{attribute 'call_after_init'}
{attribute 'reflection'}
FUNCTION_BLOCK ABSTRACT T_UnitTestBase IMPLEMENTS I_UnitTest
VAR
    {attribute 'instance-path'}
    {attribute 'no_init'}
    {attribute 'analysis' := '-33'} // Inhibit unused variable warning
    InstanceName : T_MaxString;     // Initialised with the instance name

    Project  : T_MaxString;
    Plc      : T_MaxString;
    TestName : T_MaxString;

    _TestCompleted : BOOL;
    _TestFailed    : BOOL;
    State          : INT;
    CycleCount     : UDINT;
    Retest         : BOOL;
END_VAR

METHOD AssertEquals_ANY : BOOL
VAR_INPUT
    Expected : ANY;
    Actual   : ANY;
    Message  : T_MaxString;
END_VAR
VAR
    ComparisonResult : DINT;
END_VAR
ComparisonResult := MEMCMP(pBuf1 := Expected.pValue,
                           pBuf2 := Actual.pValue,
                           n     := DINT_TO_UDINT(Actual.diSize));

IF Expected.TypeClass <> Actual.TypeClass THEN
    F_LogError(TestName, FormatStringEx1('Assertion Failed - %s', Message));
    TestFailed := TRUE;
    RETURN;

ELSIF Expected.diSize <> Actual.diSize THEN
    F_LogError(TestName, FormatStringEx1('Assertion Failed - %s', Message));
    TestFailed := TRUE;
    RETURN;

ELSIF ComparisonResult <> 0 THEN
    F_LogError(TestName, FormatStringEx1('Assertion Failed - %s', Message));
    TestFailed := TRUE;
    RETURN;
END_IF

AssertEquals_ANY := TRUE;
END_METHOD

METHOD AssertEquals_BOOL : BOOL
VAR_INPUT
    Expected : BOOL;
    Actual   : BOOL;
    Message  : T_MaxString;
END_VAR
IF Expected <> Actual THEN
    F_LogError(TestName, FormatStringEx1('Assertion Failed - %s', Message));
    TestFailed := TRUE;
    RETURN;
END_IF

AssertEquals_BOOL := TRUE;
END_METHOD

METHOD AssertEquals_BYTE : BOOL
VAR_INPUT
    Expected : BYTE;
    Actual   : BYTE;
    Message  : T_MaxString;
END_VAR
IF Expected <> Actual THEN
    F_LogError(TestName, FormatStringEx1('Assertion Failed - %s', Message));
    TestFailed := TRUE;
    RETURN;
END_IF

AssertEquals_BYTE := TRUE;
END_METHOD

METHOD AssertEquals_DINT : BOOL
VAR_INPUT
    Expected : DINT;
    Actual   : DINT;
    Message  : T_MaxString;
END_VAR
IF Expected <> Actual THEN
    F_LogError(TestName, FormatStringEx1('Assertion Failed - %s', Message));
    TestFailed := TRUE;
    RETURN;
END_IF

AssertEquals_DINT := TRUE;
END_METHOD

METHOD AssertEquals_INT : BOOL
VAR_INPUT
    Expected : INT;
    Actual   : INT;
    Message  : T_MaxString;
END_VAR
IF Expected <> Actual THEN
    F_LogError(TestName, FormatStringEx1('Assertion Failed - %s', Message));
    TestFailed := TRUE;
    RETURN;
END_IF

AssertEquals_INT := TRUE;
END_METHOD

METHOD AssertEquals_LINT : BOOL
VAR_INPUT
    Expected : LINT;
    Actual   : LINT;
    Message  : T_MaxString;
END_VAR
IF Expected <> Actual THEN
    F_LogError(TestName, FormatStringEx1('Assertion Failed - %s', Message));
    TestFailed := TRUE;
    RETURN;
END_IF

AssertEquals_LINT := TRUE;
END_METHOD

METHOD AssertEquals_LREAL : BOOL
VAR_INPUT
    Expected : LREAL;
    Actual   : LREAL;
    Delta    : LREAL;
    Message  : T_MaxString;
END_VAR
IF ABS(Expected - Actual) > Delta THEN
    F_LogError(TestName, FormatStringEx1('Assertion Failed - %s', Message));
    TestFailed := TRUE;
    RETURN;
END_IF

AssertEquals_LREAL := TRUE;
END_METHOD

METHOD AssertEquals_PVOID : BOOL
VAR_INPUT
    Expected : PVOID;
    Actual   : PVOID;
    Message  : T_MaxString;
END_VAR
IF Expected <> Actual THEN
    F_LogError(TestName, FormatStringEx1('Assertion Failed - %s', Message));
    TestFailed := TRUE;
    RETURN;
END_IF

AssertEquals_PVOID := TRUE;
END_METHOD

METHOD AssertEquals_REAL : BOOL
VAR_INPUT
    Expected : REAL;
    Actual   : REAL;
    Delta    : REAL;
    Message  : T_MaxString;
END_VAR
IF ABS(Expected - Actual) > Delta THEN
    F_LogError(TestName, FormatStringEx1('Assertion Failed - %s', Message));
    TestFailed := TRUE;
    RETURN;
END_IF

AssertEquals_REAL := TRUE;
END_METHOD

METHOD AssertEquals_STRING : BOOL
VAR_INPUT
    Expected : T_MaxString;
    Actual   : T_MaxString;
    Message   : T_MaxString;
END_VAR
IF Expected <> Actual THEN
    F_LogError(TestName, FormatStringEx1('Assertion Failed - %s', Message));
    TestFailed := TRUE;
    RETURN;
END_IF

AssertEquals_STRING := TRUE;
END_METHOD

METHOD AssertEquals_UDINT : BOOL
VAR_INPUT
    Expected : UDINT;
    Actual   : UDINT;
    Message  : T_MaxString;
END_VAR
IF Expected <> Actual THEN
    F_LogError(TestName, FormatStringEx1('Assertion Failed - %s', Message));
    TestFailed := TRUE;
    RETURN;
END_IF

AssertEquals_UDINT := TRUE;
END_METHOD

METHOD AssertEquals_UINT : BOOL
VAR_INPUT
    Expected : UINT;
    Actual   : UINT;
    Message  : T_MaxString;
END_VAR
IF Expected <> Actual THEN
    F_LogError(TestName, FormatStringEx1('Assertion Failed - %s', Message));
    TestFailed := TRUE;
    RETURN;
END_IF

AssertEquals_UINT := TRUE;
END_METHOD

METHOD AssertEquals_ULINT : BOOL
VAR_INPUT
    Expected : ULINT;
    Actual   : ULINT;
    Message  : T_MaxString;
END_VAR
IF Expected <> Actual THEN
    F_LogError(TestName, FormatStringEx1('Assertion Failed - %s', Message));
    TestFailed := TRUE;
    RETURN;
END_IF

AssertEquals_ULINT := TRUE;
END_METHOD

METHOD AssertIsFalse : BOOL
VAR_INPUT
    Condition : BOOL;
    Message   : T_MaxString;
END_VAR
IF Condition THEN
    F_LogError(TestName, FormatStringEx1('Assertion Failed - %s', Message));
    TestFailed := TRUE;
    RETURN;
END_IF

AssertIsFalse := TRUE;
END_METHOD

METHOD AssertIsTrue : BOOL
VAR_INPUT
    Condition : BOOL;
    Message   : T_MaxString;
END_VAR
IF NOT Condition THEN
    F_LogError(TestName, FormatStringEx1('Assertion Failed - %s', Message));
    TestFailed := TRUE;
    RETURN;
END_IF

AssertIsTrue := TRUE;
END_METHOD

METHOD AwaitConditionIsTrue : BOOL
VAR_INPUT
    Condition : BOOL;
	MaxCycles : UDINT;
    Message   : T_MaxString;
END_VAR
IF NOT Condition THEN
    CycleCount := CycleCount + 1; // assumes cycle count is reset before calling this method
    IF CycleCount > MaxCycles THEN
        F_LogError(TestName, FormatStringEx1('Assertion Failed - %s', Message));
        TestFailed           := TRUE;
        AwaitConditionIsTrue := TRUE;
    END_IF
    RETURN;
ELSE
    CycleCount           := 0;
    AwaitConditionIsTrue := TRUE;
END_IF
END_METHOD

PROPERTY BaseClass : I_UnitTest
GET
BaseClass := THIS^;
END_GET
END_PROPERTY

{attribute 'call_after_init'}
METHOD FINAL Init
VAR
    StringSplitter : StringSplitter;
END_VAR
StringSplitter.Init(Str := InstanceName, Delim1 := '.', Delim2 := '');

IF StringSplitter.HasMore() THEN
    Project  := StringSplitter.GetNext();
    Plc      := StringSplitter.GetNext();
    TestName := StringSplitter.GetRemainder();
ELSE
    TestName := 'Unknown Test';
END_IF

State         := 0;
TestFailed    := FALSE;
TestCompleted := FALSE;
Retest        := FALSE;
END_METHOD

PROPERTY Name : T_MaxString
GET
Name := TestName;
END_GET
END_PROPERTY

{attribute 'analysis' := '-33'} // inhibit unused variable warning
METHOD ABSTRACT RunTest
END_METHOD

PROPERTY TestCompleted : BOOL
GET // PUBLIC
TestCompleted := _TestCompleted;
END_GET
SET // PROTECTED
_TestCompleted := TestCompleted;
END_SET
END_PROPERTY

PROPERTY TestFailed : BOOL
GET // PUBLIC
TestFailed := _TestFailed;
END_GET
SET // PROTECTED
_TestFailed := TestFailed;
END_SET
END_PROPERTY

END_FUNCTION_BLOCK

(* stored: Version 1.1.0.1, ProductVersion 3.1.4024.12
   POU T_UnitTestBase: Id {db1f4e28-4a18-401b-8b29-e7f500ef63dc}, SpecialFunc None
   Folder Methods: Id {a5772276-00c5-43a4-85c1-e780c7c7de3b}
   Folder Properties: Id {eb7e9c1f-ae66-405a-820c-688b53e1a9a9}
   Method AssertEquals_ANY: Id {8c39ac6a-e3a4-4e64-8b71-f758c94e977f}
   Method AssertEquals_BOOL: Id {9b94f5a5-3f4f-4415-b23b-6241a645ab07}
   Method AssertEquals_BYTE: Id {08150b43-4ff5-4e6d-953b-1154960624e2}
   Method AssertEquals_DINT: Id {eb3056ea-2f26-4cff-a482-a3994eed33c8}
   Method AssertEquals_INT: Id {42545341-2d84-46fc-9339-3e8a2b1e71b8}
   Method AssertEquals_LINT: Id {680dbc81-25a4-4297-bce7-fc7a1394820c}
   Method AssertEquals_LREAL: Id {0e4ee858-c05e-426c-a0eb-481c1ac21bf1}
   Method AssertEquals_PVOID: Id {05e72387-7114-492d-85df-e3702e9e13b2}
   Method AssertEquals_REAL: Id {65d8a8a1-9a76-4554-b6d5-1a0075d640fb}
   Method AssertEquals_STRING: Id {922f5d37-eaf4-494b-9220-811e46507baa}
   Method AssertEquals_UDINT: Id {b4316d77-900c-4326-882d-ca3aafbaea09}
   Method AssertEquals_UINT: Id {eae747e6-05b0-4235-851e-2602e98dde70}
   Method AssertEquals_ULINT: Id {4c66f248-c3df-4371-8d92-3988dcc92ed9}
   Method AssertIsFalse: Id {f6a0ec80-6087-4cea-a1de-8b927e653068}
   Method AssertIsTrue: Id {cad875ec-dfd3-4726-81dd-a6735f47baa6}
   Method AwaitConditionIsTrue: Id {0f9e6b23-9d8e-408b-b421-7fec7bed5d6f}
   Property BaseClass: Id {b4d027a7-046f-48d1-8468-ee31a4969371}
   Get Get: Id {70254247-b8af-4d35-af04-a3ea68849a8d}
   Method Init: Id {c6c815cd-69fa-4977-953d-d0e1df3e2361}
   Property Name: Id {0404f2a6-6d2f-43ce-8288-d9af3f97471a}
   Get Get: Id {23ff53f7-40cf-4dbc-ae96-089bca3dca34}
   Method RunTest: Id {c72e0459-07ad-41cb-aa90-04d972433a01}
   Property TestCompleted: Id {2c6255e4-e476-4dee-8897-fed2ded26b5a}
   Get Get: Id {b3c15a73-0247-4742-9a74-f07336c20bf4}
   Set Set: Id {ad11a1d3-bb4b-4f00-b20e-3b78d2e07e57}
   Property TestFailed: Id {00cc0457-806b-4c3e-b342-8020d5b41549}
   Get Get: Id {aa3f4237-7e3a-4059-b45a-a9bca92ca4d4}
   Set Set: Id {2ab0aa07-ac71-4498-8066-a1ebdcc81657} *)
